Staubli VAL3: condition.pgx

public program condition(num x_nOperator, num x_nValue, string x_sItem, bool& x_bResult)
begin
  // operator
  // <> >= > < <= ==
  x_bResult=false
  //
  switch x_nOperator
    case 0
      // <>
      if isDefined(saveInOut:cCount[x_sItem])
        x_bResult=(saveInOut:cCount[x_sItem].nCount!=x_nValue)
      elseIf isDefined(saveInOut:aCount[x_sItem])
        x_bResult=(aioGet(saveInOut:aCount[x_sItem].aAio)!=x_nValue)
      endIf
    break
    case 1
      // >=
      if isDefined(saveInOut:cCount[x_sItem])
        x_bResult=(saveInOut:cCount[x_sItem].nCount>=x_nValue)
      elseIf isDefined(saveInOut:aCount[x_sItem])
        x_bResult=(aioGet(saveInOut:aCount[x_sItem].aAio)>=x_nValue)
      endIf
    break
    case 2
      // >
      if isDefined(saveInOut:cCount[x_sItem])
        x_bResult=(saveInOut:cCount[x_sItem].nCount>x_nValue)
      elseIf isDefined(saveInOut:aCount[x_sItem])
        x_bResult=(aioGet(saveInOut:aCount[x_sItem].aAio)>x_nValue)
      endIf
    break
    case 3
      // <
      if isDefined(saveInOut:cCount[x_sItem])
        x_bResult=(saveInOut:cCount[x_sItem].nCount<x_nValue)
      elseIf isDefined(saveInOut:aCount[x_sItem])
        x_bResult=(aioGet(saveInOut:aCount[x_sItem].aAio)<x_nValue)
      endIf
    break
    case 4
      // <=
      if isDefined(saveInOut:cCount[x_sItem])
        x_bResult=(saveInOut:cCount[x_sItem].nCount<=x_nValue)
      elseIf isDefined(saveInOut:aCount[x_sItem])
        x_bResult=(aioGet(saveInOut:aCount[x_sItem].aAio)<=x_nValue)
      endIf
    break
    case 5
      // ==
      if isDefined(saveInOut:cCount[x_sItem])
        x_bResult=(saveInOut:cCount[x_sItem].nCount==x_nValue)
      elseIf isDefined(saveInOut:aCount[x_sItem])
        x_bResult=(aioGet(saveInOut:aCount[x_sItem].aAio)==x_nValue)
      endIf
    break
  endSwitch
end
